# EPICS substitutions: apps/pcMonitorApp/original/PC-MONITOR1.0.2-EPICS3.14.7/iocBoot/ioc/AGADI-PC-xxxx_status.subs
file status2.template {
{ NAME    = AGADI-PC-xxxx}
}
